FUNCTION_BLOCK FB_PID_CP
VAR
	FB_SP_ROC		: FB_PID_ROC;
	tTn				: TIME;
	tTv				: TIME;
	tTd				: TIME;
	SP				: REAL;
	PV				: REAL;
	fKp				: REAL;
	LMN_ROC_OUT		: REAL;
	SP_ROC_OUT		: REAL;
	PID_OUT			: REAL;
	FB_PID			: FB_PID;
	fb1stORderFilter	: FB_1stOrderFilter;
END_VAR
VAR_INPUT
	Enable			: BOOL;
	Reset			: BOOL;
	TskCycleTime	: TIME;
	CtrlCycleTime	: TIME;
	Invers			: BOOL;
	SP_INT			: REAL;
	SP_HLM			: REAL;
	SP_LLM			: REAL;
	SP_ROC			: REAL;
	PV_IN			: REAL;
	PV_TMLAG		: REAL;
	DEADBAND		: REAL;
	fI_InnerWindow	: REAL;
	ManValue		: REAL;
	Man_On			: BOOL;
	Kp				: REAL;
	Tn				: REAL;
	Tv				: REAL;
	Td				: REAL;
	Output_Min		: REAL;
	Output_Max		: REAL;
	LMN_ROC_UP		: REAL;
	LMN_ROC_DOWN	: REAL;
	LMN_HLM			: REAL;
	LMN_LLM			: REAL;
END_VAR
VAR_OUTPUT
	LMN				: REAL;
END_VAR

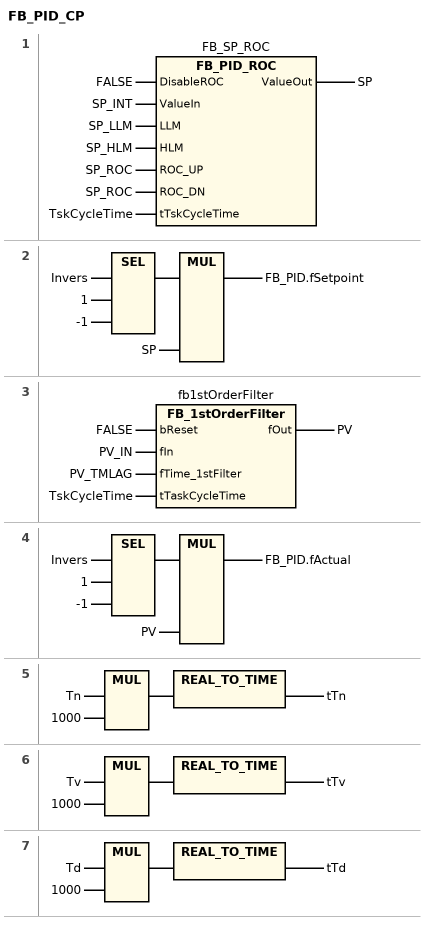
// NETWORK 1
FB_SP_ROC(
    DisableROC := FALSE,
    ValueIn := SP_INT,
    LLM := SP_LLM,
    HLM := SP_HLM,
    ROC_UP := SP_ROC,
    ROC_DN := SP_ROC,
    tTskCycleTime := TskCycleTime); // FB_PID_ROC
SP := FB_SP_ROC.ValueOut;

// NETWORK 2
FB_PID.fSetpoint := SEL(Invers, 1, -1) * SP;

// NETWORK 3
fb1stOrderFilter(bReset := FALSE, fIn := PV_IN, fTime_1stFilter := PV_TMLAG, tTaskCycleTime := TskCycleTime); // FB_1stOrderFilter
PV := fb1stOrderFilter.fOut;

// NETWORK 4
FB_PID.fActual := SEL(Invers, 1, -1) * PV;

// NETWORK 5
tTn := REAL_TO_TIME(Tn * 1000);

// NETWORK 6
tTv := REAL_TO_TIME(Tv * 1000);

// NETWORK 7
tTd := REAL_TO_TIME(Td * 1000);

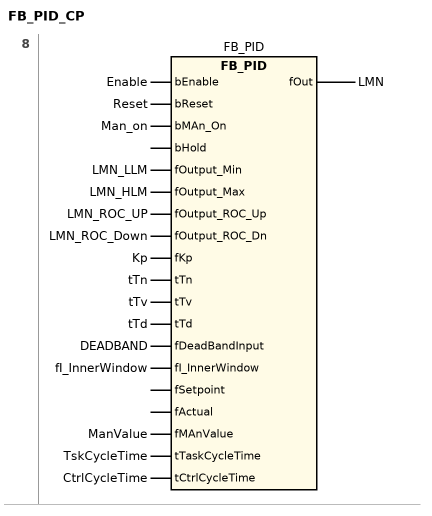
// NETWORK 8
FB_PID(
    bEnable := Enable,
    bReset := Reset,
    bMAn_On := Man_on,
    fOutput_Min := LMN_LLM,
    fOutput_Max := LMN_HLM,
    fOutput_ROC_Up := LMN_ROC_UP,
    fOutput_ROC_Dn := LMN_ROC_Down,
    fKp := Kp,
    tTn := tTn,
    tTv := tTv,
    tTd := tTd,
    fDeadBandInput := DEADBAND,
    fI_InnerWindow := fI_InnerWindow,
    fMAnValue := ManValue,
    tTaskCycleTime := TskCycleTime,
    tCtrlCycleTime := CtrlCycleTime);
LMN := FB_PID.fOut;

END_FUNCTION_BLOCK

(* stored: Version 1.1.0.1, ProductVersion 3.1.4020.12
   POU FB_PID_CP: Id {d9dcf42b-2931-4c15-afe0-72599599e35a}, SpecialFunc None *)
